Fanuc KAREL source: CA0114.KL

-- PROVISIONAL review KL for V770-1; original PC SHA256 769e956adb653a313e50e4f0462cef010ecebe68d0e933b79268bd9d1207e0d8
-- Incomplete behavior may be omitted. Consult companion uncertainty JSON. Do not deploy.
PROGRAM CA0114
%NOLOCKGROUP
BEGIN
  -- UNRESOLVED_PC offsets 0-1; opcodes 7B
  -- UNRESOLVED_PC offsets 6-16; opcodes 2D,7F
  -- UNRESOLVED_PC offsets 21-25; opcodes 7F
  -- UNRESOLVED_PC offsets 30-37; opcodes 9C,23
  -- UNRESOLVED_PC offsets 42-49; opcodes 9D,23
  -- UNRESOLVED_PC offsets 54-65; opcodes 2E,23
  -- UNRESOLVED_PC offsets 70-77; opcodes 9D,23
  -- UNRESOLVED_PC offsets 82-91; opcodes 3F,75
  -- UNRESOLVED_PC offsets 96-110; opcodes 2E,22,9D,33,35
  -- UNRESOLVED_PC offsets 115-129; opcodes 2E,22,9D,33,35
  -- UNRESOLVED_PC offsets 134-149; opcodes 2E,22,32,35
  -- UNRESOLVED_PC offsets 154-169; opcodes 2E,22,32,35
  -- UNRESOLVED_PC offsets 174-232; opcodes 27,22,22,22,22,22,22,22,22,AA,23
  -- UNRESOLVED_PC offsets 237-241; opcodes 7F
END CA0114
